(* CODESYS project TestModbus.project
   Title: TestModbus
   Version: 0.0.0.0
   Author: Peter

Project tree, tasks and I/O mapping:
  MyController : TM241CEC24T/U, Schneider Electric, order no. TM241CEC24T/U, version 4.0.6.18
    application Application
      task MAST (cyclic, interval 20 ms, priority 15, watchdog 100 ms x 1) calls nothing
      global variables GVL
    DI : Digital Inputs, Schneider Electric, version 4.0.6.18
        input  iwDI_IW0 : WORD  // IW0
        input  ibDI_IB1 : BYTE  // IB1
    DQ : Digital Outputs, Schneider Electric, version 4.0.6.18
        output qwDQ_QW0 : WORD  // QW0
        output qbDQ_QB1 : BYTE  // QB1
    Counters : Counters, Schneider Electric, version 4.0.6.18
    Pulse_Generators : Pulse Generators, Schneider Electric, version 4.0.6.18
    Cartridge_1 : Cartridge, Schneider Electric, version 4.0.6.18
    IO_Bus : IO bus - TM3, Schneider Electric, version 4.0.6.18
      Module_1 : TM3AQ2/G, Schneider Electric, order no. TM3AQ2/G, version 1.0.0.12
          output qiModule_1_QW0 : INT  // QW0
          output qiModule_1_QW1 : INT  // QW1
          input  ibModule_1_IBStatusQW0 : BYTE  // IBStatusQW0
          input  ibModule_1_IBStatusQW1 : BYTE  // IBStatusQW1
      Module_2 : TM3SAF5R/G, Schneider Electric, order no. TM3SAF5R/G, version 1.0.1.12
          input  iwModule_2_IW0 : WORD  // IW0
          output qbModule_2_QB0 : BYTE  // QB0
    COM_Bus : COM bus, Schneider Electric, version 4.0.6.18
    Ethernet_1 : Ethernet Network, Schneider Electric, version 4.0.6.18
    Serial_Line_1 : Serial line, Schneider Electric, version 4.0.6.18
      SoMachine_Network_Manager : SoMachine-Network Manager, Schneider Electric, version 4.0.0.2
    Serial_Line_2 : Serial line, Schneider Electric, version 4.0.6.18
      Modbus_Manager : Modbus Manager, Schneider Electric, version 4.0.0.2
    CAN_1 : CANopen bus, Schneider Electric, version 4.0.6.18
*)

// MyController/Application/GVL
VAR_GLOBAL
END_VAR
